// TIA Portal V15.1 export
// export: Created 2024-06-21T08:41:08.2360509Z, ExportSetting WithDefaults, DisplayName Totally Integrated Automation Portal, DisplayVersion V15.1 Update 5, DisplayName TIA Portal Openness, DisplayVersion V15.1 Update 5, DisplayName SINAMICS Startdrive Advanced, DisplayVersion V15.1, DisplayName G130, G150, S120, S150, SINAMICS MV, S210, DisplayVersion V15.1, DisplayName G110M, G120, G120C, G120D, G120P, DisplayVersion V15.1, DisplayName STEP 7 Professional, DisplayVersion V15.1 Update 5, DisplayName STEP 7 Safety, DisplayVersion V15.1, DisplayName WinCC Professional, DisplayVersion V15.1 Update 5, DisplayName SIMATIC Visualization Architect, DisplayVersion V15.1
FUNCTION_BLOCK "LGBBodyStopperSub"   // FB6667, SCL
TITLE = LBodyTypeSimSub
{ S7_Optimized_Access := 'FALSE' }
AUTHOR : IMTECH
VERSION : 1.0
// stored: AutoNumber false, IsIECCheckEnabled false, SetENOAutomatically False, UDAEnableTagReadback false
   VAR_INPUT
      I_BodyNr { ExternalAccessible := 'False'; ExternalVisible := 'False'; ExternalWritable := 'False'} : DInt;
      I_ColorCodeBC { ExternalAccessible := 'False'; ExternalVisible := 'False'; ExternalWritable := 'False'} : DInt;
      I_ColorCodeCC { ExternalAccessible := 'False'; ExternalVisible := 'False'; ExternalWritable := 'False'} : DInt;
      I_MMFRUSS { ExternalAccessible := 'False'; ExternalVisible := 'False'; ExternalWritable := 'False'} : DInt;
      I_MM { ExternalAccessible := 'False'; ExternalVisible := 'False'; ExternalWritable := 'False'} : Int;
      I_R { ExternalAccessible := 'False'; ExternalVisible := 'False'; ExternalWritable := 'False'} : Int;
      I_S2 { ExternalAccessible := 'False'; ExternalVisible := 'False'; ExternalWritable := 'False'} : Int;
      I_StartSearch { ExternalAccessible := 'False'; ExternalVisible := 'False'; ExternalWritable := 'False'} : Bool;
      I_ClearSearch { ExternalAccessible := 'False'; ExternalVisible := 'False'; ExternalWritable := 'False'} : Bool;
      I_HMICmdForce { ExternalAccessible := 'False'; ExternalVisible := 'False'; ExternalWritable := 'False'} : Bool;
      I_HMICmdJustR { ExternalAccessible := 'False'; ExternalVisible := 'False'; ExternalWritable := 'False'} : Bool;
      I_HMICmdJustS2 { ExternalAccessible := 'False'; ExternalVisible := 'False'; ExternalWritable := 'False'} : Bool;
      I_HMICmdMM1stLayer { ExternalAccessible := 'False'; ExternalVisible := 'False'; ExternalWritable := 'False'} : Bool;
      I_HMICmdMM2ndLayer { ExternalAccessible := 'False'; ExternalVisible := 'False'; ExternalWritable := 'False'} : Bool;
   END_VAR
   VAR_OUTPUT
      O_BodyGo { ExternalAccessible := 'False'; ExternalVisible := 'False'; ExternalWritable := 'False'} : Bool;
      O_BodyStop { ExternalAccessible := 'False'; ExternalVisible := 'False'; ExternalWritable := 'False'} : Bool;
      O_Status_HMICmdForce { ExternalAccessible := 'False'; ExternalVisible := 'False'; ExternalWritable := 'False'} : Bool;
      O_Status_HMICmdMM1stLayer { ExternalAccessible := 'False'; ExternalVisible := 'False'; ExternalWritable := 'False'} : Bool;
      O_Status_HMICmdMM2ndLayer { ExternalAccessible := 'False'; ExternalVisible := 'False'; ExternalWritable := 'False'} : Bool;
      O_Status_TABGeneral { ExternalAccessible := 'False'; ExternalVisible := 'False'; ExternalWritable := 'False'} : Bool;
      O_Status_TABSealing { ExternalAccessible := 'False'; ExternalVisible := 'False'; ExternalWritable := 'False'} : Bool;
      O_Status_TABPaint { ExternalAccessible := 'False'; ExternalVisible := 'False'; ExternalWritable := 'False'} : Bool;
      O_Status_BodyNr { ExternalAccessible := 'False'; ExternalVisible := 'False'; ExternalWritable := 'False'} : Array[1..10] of Bool;
      O_Status_ColorCodeBC { ExternalAccessible := 'False'; ExternalVisible := 'False'; ExternalWritable := 'False'} : Array[1..10] of Bool;
      O_Status_ColorCodeCC { ExternalAccessible := 'False'; ExternalVisible := 'False'; ExternalWritable := 'False'} : Array[1..10] of Bool;
      O_Status_MM { ExternalAccessible := 'False'; ExternalVisible := 'False'; ExternalWritable := 'False'} : Array[1..10] of Bool;
      O_Status_MMwithR { ExternalAccessible := 'False'; ExternalVisible := 'False'; ExternalWritable := 'False'} : Array[1..10] of Bool;
      O_Status_MMwithS2 { ExternalAccessible := 'False'; ExternalVisible := 'False'; ExternalWritable := 'False'} : Array[1..10] of Bool;
      O_AC_BodyStop { ExternalAccessible := 'False'; ExternalVisible := 'False'; ExternalWritable := 'False'} : Bool;
   END_VAR
   VAR_IN_OUT
      IO_ArrayHMI_BodyNr : Array[1..10] of DInt;
      IO_ArrayHMI_ColorCodeBC : Array[1..10] of Int;
      IO_ArrayHMI_ColorCodeCC : Array[1..10] of Int;
      IO_ArrayHMI_MM : Array[1..10] of Int;
      IO_ArrayHMI_MMwithR : Array[1..10] of Int;
      IO_ArrayHMI_MMwithS2 : Array[1..10] of Int;
      IO_ArrayHMI_R : Array[1..10] of Int;
      IO_ArrayHMI_S2 : Array[1..10] of Int;
      IO_ArrayHMI_DuoTone : Array[1..10] of Int;
   END_VAR
   VAR DB_SPECIFIC
      Index { ExternalAccessible := 'False'; ExternalVisible := 'False'; ExternalWritable := 'False'} : Int;
      BodyGo { ExternalAccessible := 'False'; ExternalVisible := 'False'; ExternalWritable := 'False'} : Bool;
      BodyStop { ExternalAccessible := 'False'; ExternalVisible := 'False'; ExternalWritable := 'False'} : Bool;
      NewBodyNr { ExternalAccessible := 'False'; ExternalVisible := 'False'; ExternalWritable := 'False'} : DInt;
      NewColorCodeBC { ExternalAccessible := 'False'; ExternalVisible := 'False'; ExternalWritable := 'False'} : DInt;
      NewColorCodeCC { ExternalAccessible := 'False'; ExternalVisible := 'False'; ExternalWritable := 'False'} : DInt;
      NewMMFRUSS { ExternalAccessible := 'False'; ExternalVisible := 'False'; ExternalWritable := 'False'} : DInt;
      Status_HMICmdForce { ExternalAccessible := 'False'; ExternalVisible := 'False'; ExternalWritable := 'False'} : Bool;
      Status_HMICmdMM1stLayer { ExternalAccessible := 'False'; ExternalVisible := 'False'; ExternalWritable := 'False'} : Bool;
      Status_HMICmdMM2ndLayer { ExternalAccessible := 'False'; ExternalVisible := 'False'; ExternalWritable := 'False'} : Bool;
      Status_TABGeneral { ExternalAccessible := 'False'; ExternalVisible := 'False'; ExternalWritable := 'False'} : Bool;
      Status_TABSealing { ExternalAccessible := 'False'; ExternalVisible := 'False'; ExternalWritable := 'False'} : Bool;
      Status_TABPaint { ExternalAccessible := 'False'; ExternalVisible := 'False'; ExternalWritable := 'False'} : Bool;
      Status_BodyNr { ExternalAccessible := 'False'; ExternalVisible := 'False'; ExternalWritable := 'False'} : Array[1..10] of Bool;
      Status_ColorCodeBC { ExternalAccessible := 'False'; ExternalVisible := 'False'; ExternalWritable := 'False'} : Array[1..10] of Bool;
      Status_ColorCodeCC { ExternalAccessible := 'False'; ExternalVisible := 'False'; ExternalWritable := 'False'} : Array[1..10] of Bool;
      Status_MM { ExternalAccessible := 'False'; ExternalVisible := 'False'; ExternalWritable := 'False'} : Array[1..10] of Bool;
      Status_MMwithR { ExternalAccessible := 'False'; ExternalVisible := 'False'; ExternalWritable := 'False'} : Array[1..10] of Bool;
      Status_MMwithS2 { ExternalAccessible := 'False'; ExternalVisible := 'False'; ExternalWritable := 'False'} : Array[1..10] of Bool;
      FlankHMICmdForce { ExternalAccessible := 'False'; ExternalVisible := 'False'; ExternalWritable := 'False'} : Bool;
      AlarmBodyStop { ExternalAccessible := 'False'; ExternalVisible := 'False'; ExternalWritable := 'False'} : Bool;
   END_VAR
   VAR_TEMP
      NotUsedBool : Bool;
      NotUsedInt : Int;
      NotUsedWord : Word;
      NotUsedDWord : DWord;
   END_VAR
BEGIN
   //************************************
   //*                                  *
   //*             LOGIC FB             *
   //*                                  *
   //************************************

   // CLEAR SEARCH FUNCTION
   IF #I_ClearSearch OR (#I_BodyNr = 0) OR (#I_MMFRUSS = 0) OR (#I_BodyNr <> #NewBodyNr) OR (#I_ColorCodeBC <> #NewColorCodeBC) OR (#I_ColorCodeCC <> #NewColorCodeCC) OR (#I_MMFRUSS <> #NewMMFRUSS) THEN
       #Index := 1;
       WHILE #Index <= 10 DO
           #Status_BodyNr[#Index] := False;
           #Status_ColorCodeBC[#Index] := False;
           #Status_ColorCodeCC[#Index] := False;
           #Status_MM[#Index] := False;
           #Status_MMwithR[#Index] := False;
           #Status_MMwithS2[#Index] := False;
           #Index := #Index + 1;
       END_WHILE;
       #BodyGo := False;
       #BodyStop := False;
       #AlarmBodyStop := False;
       #Status_HMICmdForce := False;
       #Status_HMICmdMM1stLayer := False;
       #Status_HMICmdMM2ndLayer := False;
       #Status_TABGeneral := False;
       #Status_TABSealing := False;
       #Status_TABPaint := False;
       #NewBodyNr := #I_BodyNr;
       #NewColorCodeBC := #I_ColorCodeBC;
       #NewColorCodeCC := #I_ColorCodeCC;
       #NewMMFRUSS := #I_MMFRUSS;
   END_IF;

   // BODY NOT OK ---> Something is wrong ...
   IF #I_StartSearch AND #I_BodyNr <> #NewBodyNr AND ((#I_BodyNr = 0) OR (#I_MMFRUSS = 0) OR (#I_ColorCodeBC = 0) OR (#I_ColorCodeCC = 0)) THEN
       #BodyStop := True;
       #AlarmBodyStop := True;
   END_IF;

   // STATUS HmiCmd Force -> Indicator that the selection is activ
       IF NOT #I_HMICmdForce THEN #FlankHMICmdForce:= False; END_IF;    

       IF #I_HMICmdForce AND (#I_BodyNr <> 0) AND (#I_MMFRUSS <> 0) AND #AlarmBodyStop AND NOT #FlankHMICmdForce THEN
           IF NOT #Status_HMICmdForce THEN
               #Status_HMICmdForce:= True;
           ELSE
               #Status_HMICmdForce:= False;           
           END_IF;
           #FlankHMICmdForce:= True;
       END_IF;

   // SEARCH IN THE LIST ---> BodyNr - MM - MM with S2 - ColorCode      
       IF #I_StartSearch AND (#I_BodyNr <> 0) AND (#I_ColorCodeBC <> 0) AND (#I_ColorCodeCC <> 0) AND (#I_MMFRUSS <> 0) AND NOT #BodyGo AND NOT #BodyStop THEN
           // BodyNr
           #Index:= 1;
           WHILE (#Index <= 10) DO
               IF #I_BodyNr = #IO_ArrayHMI_BodyNr[#Index] THEN
                   #Status_BodyNr[#Index] := True;
                   #BodyStop := True;
                   #AlarmBodyStop := True;
                   #Status_TABGeneral := True;
               END_IF;
               #Index := #Index + 1;
           END_WHILE;

           // MM
           #Index:= 1;
           WHILE (#Index <= 10) DO
               IF (#I_MM = #IO_ArrayHMI_MM[#Index]) THEN
                   #Status_MM[#Index]:= True;
                   #BodyStop:= True;
                   #AlarmBodyStop:= True;
                   #Status_TABGeneral := True;
               END_IF;
               #Index:= #Index + 1;
           END_WHILE;

           // MM with S2
           #Index:= 1;
           WHILE (#Index <= 10) AND NOT #I_HMICmdJustS2 DO
               IF (#I_MM = #IO_ArrayHMI_MMwithS2[#Index]) AND (#I_S2 = #IO_ArrayHMI_S2[#Index]) THEN
                   #Status_MMwithS2[#Index]:= True;
                   #BodyStop:= True;
                   #AlarmBodyStop:= True;
                   #Status_TABGeneral := True;
               END_IF;
               #Index:= #Index + 1;
           END_WHILE;
           #Index:= 1;
           WHILE (#Index <= 10) AND #I_HMICmdJustS2 DO
               IF (#I_S2 = #IO_ArrayHMI_S2[#Index]) THEN
                   #Status_MMwithS2[#Index] := True;
                   #BodyStop := True;
                   #AlarmBodyStop := True;
                   #Status_TABGeneral := True;
               END_IF;
               #Index:= #Index + 1;
           END_WHILE;

           // MM with R
           #Index := 1;
           WHILE (#Index <= 10) AND NOT #I_HMICmdJustR DO
               IF (#I_MM = #IO_ArrayHMI_MMwithR[#Index]) AND (#I_R = #IO_ArrayHMI_R[#Index]) THEN
                   #Status_MMwithR[#Index] := True;
                   #BodyStop := True;
                   #AlarmBodyStop := True;
                   #Status_TABGeneral := True;
               END_IF;
               #Index := #Index + 1;
           END_WHILE;
           #Index := 1;
           WHILE (#Index <= 10) AND #I_HMICmdJustR DO
               IF (#I_R = #IO_ArrayHMI_R[#Index]) THEN
                   #Status_MMwithR[#Index] := True;
                   #BodyStop := True;
                   #AlarmBodyStop := True;
                   #Status_TABGeneral := True;
               END_IF;
               #Index := #Index + 1;
           END_WHILE;

           // ColorCode
               // BC
           #Index := 1;
           WHILE (#Index <= 10) AND (#I_ColorCodeBC > 1000) DO // Color Code = YXXX
               IF (#I_ColorCodeBC = #IO_ArrayHMI_ColorCodeBC[#Index] + #IO_ArrayHMI_DuoTone[#Index]) THEN
                   #Status_ColorCodeBC[#Index] := True;
                   #BodyStop := True;
                   #AlarmBodyStop := True;
                   #Status_TABPaint := True;
               END_IF;
               #Index := #Index + 1;
           END_WHILE;
           #Index := 1;
           WHILE (#Index <= 10) AND (#I_ColorCodeBC < 1000) DO // Color Code = XXX
               IF (#I_ColorCodeBC + 9000 = #IO_ArrayHMI_ColorCodeBC[#Index] + #IO_ArrayHMI_DuoTone[#Index]) THEN
                   #Status_ColorCodeBC[#Index] := True;
                   #BodyStop := True;
                   #AlarmBodyStop := True;
                   #Status_TABPaint := True;
               END_IF;
               #Index := #Index + 1;
           END_WHILE;
           IF (1 = #I_ColorCodeBC / 1000) AND #I_HMICmdMM1stLayer THEN  // Extra Button "1stLayer"
               #Status_HMICmdMM1stLayer := True;
               #BodyStop := True;
               #AlarmBodyStop := True;
               #Status_TABPaint := True;
           END_IF;
           IF (2 = #I_ColorCodeBC / 1000) AND #I_HMICmdMM2ndLayer THEN  // Extra Button "2ndLayer"
               #Status_HMICmdMM2ndLayer := True;
               #BodyStop := True;
               #AlarmBodyStop := True;
               #Status_TABPaint := True;
           END_IF;
               // CC
           #Index := 1;
           WHILE (#Index <= 10) DO
               IF (#I_ColorCodeCC) = #IO_ArrayHMI_ColorCodeCC[#Index] THEN
                   #Status_ColorCodeCC[#Index] := True;
                   #BodyStop := True;
                   #AlarmBodyStop := True;
                   #Status_TABPaint := True;
               END_IF;
               #Index := #Index + 1;
           END_WHILE;

           // Body is ok
           IF NOT #BodyStop THEN
               #BodyGo:= True;   
           END_IF;    
       END_IF;       

   // FORCE A BODY
       IF #BodyStop AND #Status_HMICmdForce THEN
           #BodyGo := True;
           #BodyStop := False;
           #AlarmBodyStop := False;
           #Status_TABGeneral := False;
           #Status_TABSealing := False;
           #Status_TABPaint := False;
       END_IF;

   // OUTPUT
       #O_BodyGo:= #BodyGo;
       #O_BodyStop:= #BodyStop;
       #O_Status_HMICmdForce := #Status_HMICmdForce;
       #O_Status_HMICmdMM1stLayer := #Status_HMICmdMM1stLayer;
       #O_Status_HMICmdMM2ndLayer := #Status_HMICmdMM2ndLayer;
       #O_Status_BodyNr:= #Status_BodyNr;
       #O_Status_ColorCodeBC := #Status_ColorCodeBC;
       #O_Status_ColorCodeCC := #Status_ColorCodeCC;
       #O_Status_MM := #Status_MM;
       #O_Status_MMwithR := #Status_MMwithR;
       #O_Status_MMwithS2:= #Status_MMwithS2;
       #O_Status_TABGeneral := #Status_TABGeneral;
       #O_Status_TABSealing := #Status_TABSealing;
       #O_Status_TABPaint := #Status_TABPaint;
       #O_AC_BodyStop:= #AlarmBodyStop;
END_FUNCTION_BLOCK
